FUNCTION_BLOCK AlarmLogger IMPLEMENTS IVisitor
VAR
	_value: REAL;
END_VAR

PROPERTY actualValue : REAL
GET
ActualValue:=this^._value;
END_GET
END_PROPERTY

METHOD updateValue : REAL
VAR_INPUT
	value: REAL;
END_VAR
this^._value:= value;
END_METHOD

END_FUNCTION_BLOCK

(* stored: Version 1.1.0.1
   POU AlarmLogger: Id {ba3262ee-64d9-4706-8b90-95ee0e106f53}, SpecialFunc None
   Property actualValue: Id {92d1fb36-0f53-4507-91df-0802767ffdde}
   Get Get: Id {991cfbcb-80d4-41c7-8de3-ee61721d55a0}
   Method updateValue: Id {d597d421-924b-4546-8b84-e80b8a4d853a} *)
